{attribute addProperty BoxType "EL3111-0000-0016"}
{attribute addProperty Id "AI_StandardAT %I*AI_Standard_904746A23240WcStateAT %I*WcState_F855686C1620InfoDataAT %I*InfoData_BC63D37F80100"}
{attribute addProperty CRC "2663782158"}
{attribute addProperty SizeInBites "128"}
{attribute addProperty SizeInBytes "16"}
TYPE EL3111_EA8DF7B0 :
STRUCT
	{attribute addProperty Name "AI_Standard"}
	AI_Standard : AI_Standard_904746A2;
	{attribute addProperty Name "WcState"}
	WcState : WcState_F855686C;
	{attribute addProperty Name "InfoData"}
	InfoData : InfoData_BC63D37F;
END_STRUCT
END_TYPE

(* stored: Version 1.2.0.0, ProductVersion 3.1.4024.9
   DUT EL3111_EA8DF7B0: Id {977d872f-cd9d-4a32-8e6b-e92e7a487932} *)
